{attribute 'TcGenerated'}
{attribute 'no-analysis'}
{attribute 'linkalways'}
// This function has been automatically generated from the project information.
VAR_GLOBAL CONSTANT
    {attribute 'const_non_replaced'}
    stLibVersion_PMPS : ST_LibVersion := (iMajor := 3, iMinor := 14, iBuild := 0, iRevision := 0, nFlags := 1, sVersion := '3.14.0');
END_VAR

(* stored: Version 1.1.0.1, ProductVersion 3.1.4022.18
   GVL Global_Version: Id {3e8b0d67-4380-4e91-81ec-b8b82dca4df4} *)
